SUBAPPLICATION AE2_ILOCK_T_FF_TO_AX (* Ein Kettenglied eines wechselseitig verriegelten Toggle-Flip-Flops via AE2-Bidirektional-Adapter (SOCKET/PLUG-Kette), Ausgang als AX-Adapter. Generisch fuer beliebig viele Teilnehmer nutzbar, indem PLUG des einen an SOCKET des naechsten angeschlossen wird - jeder Klick verriegelt die uebrigen Glieder der Kette gegenseitig (nur ein Ausgang gleichzeitig aktiv). *)
  (* Standard: 61499-2 *)
  (* Version 1.0, 2026-09-09, Franz Höpfinger, Meisterschulen am Ostbahnhof, Ausgelagert aus Uebung_004b4c_AX (Uebung_004b4c_sub_AE) zur Wiederverwendung fuer weitere verriegelte Toggle-Ketten. *)
  PACKAGE MyLib::sys;
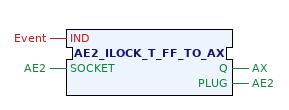
  EVENT_INPUT
    IND;
  END_EVENT
  SOCKETS
    SOCKET : adapter::types::bidirectional::AE2;
  END_SOCKETS
  PLUGS
    Q : adapter::types::unidirectional::AX;
    PLUG : adapter::types::bidirectional::AE2;
  END_PLUGS
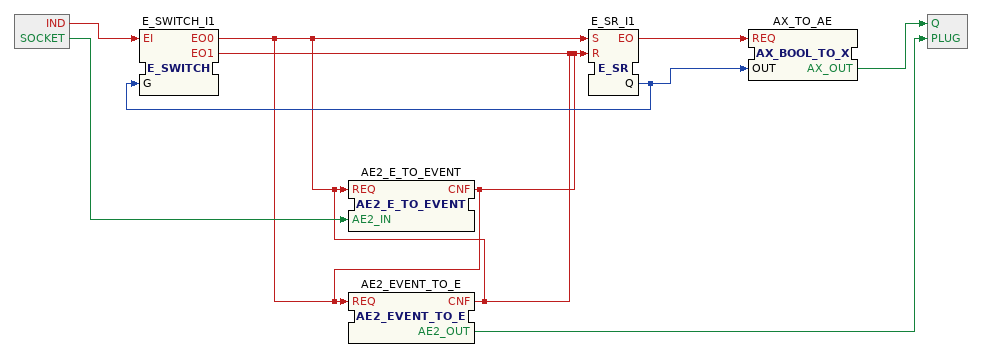
  FBS
    E_SR_I1 : iec61499::events::E_SR;
    E_SWITCH_I1 : iec61499::events::E_SWITCH;
    AE2_EVENT_TO_E : adapter::conversion::bidirectional::AE2_EVENT_TO_E;
    AE2_E_TO_EVENT : adapter::conversion::bidirectional::AE2_E_TO_EVENT;
    AX_TO_AE : adapter::conversion::unidirectional::AX_BOOL_TO_X;
  END_FBS
  EVENT_CONNECTIONS
    E_SWITCH_I1.EO0 TO E_SR_I1.S;
    E_SWITCH_I1.EO1 TO E_SR_I1.R;
    IND TO E_SWITCH_I1.EI;
    E_SWITCH_I1.EO0 TO AE2_EVENT_TO_E.REQ;
    AE2_E_TO_EVENT.CNF TO E_SR_I1.R;
    AE2_EVENT_TO_E.CNF TO E_SR_I1.R;
    E_SWITCH_I1.EO0 TO AE2_E_TO_EVENT.REQ;
    E_SR_I1.EO TO AX_TO_AE.REQ;
    AE2_E_TO_EVENT.CNF TO AE2_EVENT_TO_E.REQ;
    AE2_EVENT_TO_E.CNF TO AE2_E_TO_EVENT.REQ;
  END_CONNECTIONS
  DATA_CONNECTIONS
    E_SR_I1.Q TO E_SWITCH_I1.G;
    E_SR_I1.Q TO AX_TO_AE.OUT;
  END_CONNECTIONS
  ADAPTER_CONNECTIONS
    SOCKET TO AE2_E_TO_EVENT.AE2_IN;
    AE2_EVENT_TO_E.AE2_OUT TO PLUG;
    AX_TO_AE.AX_OUT TO Q;
  END_CONNECTIONS
END_SUBAPPLICATION
